// TIA Portal V18 export
VAR_GLOBAL   // PLC tag table "S1_R2"
   S1_R2_Valve_Up AT %Q400.0 : Bool;
   S1_R2_Valve_Down AT %Q400.1 : Bool;
   S1_R2_Sen_Drv_1 AT %Q400.2 : Bool;
   S1_R2_Sen_Drv_2 AT %Q400.3 : Bool;
   S1_R2_Sen_Drv_3 AT %Q400.4 : Bool;
   S1_R2_Sen_Drv_4 AT %Q400.5 : Bool;
   S1_R2_Sen_Val1_Up AT %Q400.6 : Bool;
   S1_R2_Sen_Val1_Down AT %Q400.7 : Bool;
   S1_R2_Sen_Val2_Up AT %Q401.0 : Bool;
   S1_R2_Sen_Val2_Down AT %Q401.1 : Bool;
   S1_R2_Hyd_Filtr AT %Q401.2 : Bool;
   S1_R2_Hyd_Empty AT %Q401.3 : Bool;
   S1_R2_Safety1_1 AT %I450.0 : Bool;
   S1_R2_Safety2_1 AT %I450.1 : Bool;
   S1_R2_Safety3_1 AT %I450.2 : Bool;
   S1_R2_Safety4_1 AT %I450.3 : Bool;
   S1_R2_Safety1_2 AT %I451.0 : Bool;
   S1_R2_Safety2_2 AT %I451.1 : Bool;
   S1_R2_Safety3_2 AT %I451.2 : Bool;
   S1_R2_Safety4_2 AT %I451.3 : Bool;
END_VAR
